ABB RAPID module: tester_right.mod

MODULE tester_right
LOCAL CONST string YuMi_App_Program_Version:="1.0.1"; !Do not edit or remove this line!
LOCAL VAR robtarget s35 := [[358.37,-68.33,133],[0.275214,0.0426853,0.863133,0.421233],[0,-2,-1,11],[-117.324,9E+09,9E+09,9E+09,9E+09,9E+09]];
LOCAL VAR robtarget s34 := [[537.58,-221.99,107.92],[0.0203865,-0.290011,-0.954645,-0.0642686],[0,-2,0,11],[-176.329,9E+09,9E+09,9E+09,9E+09,9E+09]];
LOCAL VAR robtarget s33 := [[467.55,-213.81,57.09],[0.496621,-0.80295,-0.0521253,-0.325456],[0,0,0,11],[165.649,9E+09,9E+09,9E+09,9E+09,9E+09]];
LOCAL VAR robtarget s32 := [[306.2,-52.91,16.67],[0.717218,-0.691447,0.0462227,-0.073234],[1,0,0,11],[153.702,9E+09,9E+09,9E+09,9E+09,9E+09]];
LOCAL VAR robtarget s31 := [[310.32,9.22,5.39],[0.716537,-0.693105,0.0533556,-0.0577434],[1,0,0,11],[153.592,9E+09,9E+09,9E+09,9E+09,9E+09]];
LOCAL VAR robtarget s30 := [[306.4,0.86,31.28],[0.734937,-0.673984,0.0222505,-0.0715334],[1,0,0,11],[152.628,9E+09,9E+09,9E+09,9E+09,9E+09]];
LOCAL VAR robtarget s29 := [[311.66,-63,44.82],[0.56004,-0.794065,-0.0460185,-0.231728],[0,0,0,11],[154.727,9E+09,9E+09,9E+09,9E+09,9E+09]];
LOCAL VAR robtarget s28 := [[299.07,-103.69,-6.2],[0.280816,-0.867914,-0.384884,-0.140468],[0,0,-1,11],[154.742,9E+09,9E+09,9E+09,9E+09,9E+09]];
LOCAL VAR robtarget s27 := [[352.75,-152.26,-47.58],[0.00513543,0.702291,0.711785,0.0111369],[1,0,-1,1010],[149.493,9E+09,9E+09,9E+09,9E+09,9E+09]];
LOCAL VAR robtarget s26 := [[345.22,-148.03,-90.26],[0.00526599,-0.716656,-0.697243,-0.0151133],[1,0,-1,1010],[153.525,9E+09,9E+09,9E+09,9E+09,9E+09]];
LOCAL VAR robtarget s25 := [[345.92,-149.32,-76.57],[0.0108524,-0.753223,-0.657389,-0.0194125],[1,0,-1,1010],[156.115,9E+09,9E+09,9E+09,9E+09,9E+09]];
LOCAL VAR robtarget s24 := [[357.66,-150.93,-35.49],[0.00970556,0.737723,0.663169,0.126002],[0,0,0,1010],[163.101,9E+09,9E+09,9E+09,9E+09,9E+09]];
LOCAL VAR robtarget s23 := [[388.73,-144.04,35.15],[0.0733127,-0.627707,-0.616071,-0.470176],[0,-1,0,11],[-163.98,9E+09,9E+09,9E+09,9E+09,9E+09]];
LOCAL VAR robtarget s22 := [[342.3,-148.5,49.05],[0.350551,-0.529329,-0.492073,-0.595641],[0,-1,0,11],[-159.838,9E+09,9E+09,9E+09,9E+09,9E+09]];
LOCAL VAR robtarget s21 := [[285.33,-50.36,-15.16],[0.467312,-0.523371,-0.473345,-0.532585],[0,-1,0,11],[-169.176,9E+09,9E+09,9E+09,9E+09,9E+09]];
LOCAL VAR robtarget s20 := [[284.5,11.38,-19.53],[0.493118,-0.506889,-0.461514,-0.535634],[1,-1,0,11],[-170.503,9E+09,9E+09,9E+09,9E+09,9E+09]];
LOCAL VAR robtarget s19 := [[284.5,11.39,-19.53],[0.49312,-0.506885,-0.461513,-0.535636],[1,-1,0,11],[-170.503,9E+09,9E+09,9E+09,9E+09,9E+09]];
LOCAL VAR robtarget s18 := [[283.93,11.08,-19.46],[0.493586,-0.506785,-0.461377,-0.535419],[1,-1,0,11],[-170.522,9E+09,9E+09,9E+09,9E+09,9E+09]];
LOCAL VAR robtarget s17 := [[283.93,11.07,-19.46],[0.493582,-0.506788,-0.461378,-0.535418],[1,-1,0,11],[-170.522,9E+09,9E+09,9E+09,9E+09,9E+09]];
LOCAL VAR robtarget s16 := [[283.93,11.07,-19.47],[0.493573,-0.5068,-0.461384,-0.53541],[1,-1,0,11],[-170.522,9E+09,9E+09,9E+09,9E+09,9E+09]];
LOCAL VAR robtarget s15 := [[282.43,12.65,-10.4],[0.493036,-0.507364,-0.460348,-0.536261],[1,-1,0,11],[-169.512,9E+09,9E+09,9E+09,9E+09,9E+09]];
LOCAL VAR robtarget s14 := [[285.29,11.12,13.96],[0.483333,-0.506561,-0.479515,-0.529009],[0,-1,0,11],[-167.842,9E+09,9E+09,9E+09,9E+09,9E+09]];
LOCAL VAR robtarget s13 := [[299.2,-72.45,52.01],[0.505778,-0.516645,-0.4521,-0.522371],[0,-1,0,11],[-163.463,9E+09,9E+09,9E+09,9E+09,9E+09]];
LOCAL VAR robtarget s12 := [[301.58,-60.87,67.73],[0.531821,-0.485612,-0.484682,-0.496418],[0,-1,0,11],[-162.383,9E+09,9E+09,9E+09,9E+09,9E+09]];
LOCAL VAR robtarget s11 := [[315.49,-68.53,58.63],[0.496532,-0.515442,-0.489328,-0.49833],[0,-1,0,11],[-161.717,9E+09,9E+09,9E+09,9E+09,9E+09]];
LOCAL VAR robtarget s10 := [[315.48,-68.53,58.63],[0.496531,-0.515444,-0.489327,-0.49833],[0,-1,0,11],[-161.717,9E+09,9E+09,9E+09,9E+09,9E+09]];
LOCAL VAR robtarget s9 := [[335.43,-129.87,89.3],[0.417557,-0.554213,-0.666307,-0.273002],[0,-1,0,11],[-161.728,9E+09,9E+09,9E+09,9E+09,9E+09]];
LOCAL VAR robtarget s8 := [[345.66,-189.94,55.79],[0.0163252,-0.262519,-0.955378,-0.134427],[0,-2,0,11],[-147.912,9E+09,9E+09,9E+09,9E+09,9E+09]];
LOCAL VAR robtarget s7 := [[253.69,-227.69,32.72],[0.0393185,-0.0503203,0.995728,-0.0666949],[0,-2,0,11],[-149.635,9E+09,9E+09,9E+09,9E+09,9E+09]];
LOCAL VAR robtarget s6 := [[285.53,-146.72,-90.22],[0.000644566,7.67705E-05,-0.999188,0.0402885],[0,-2,0,11],[-155.028,9E+09,9E+09,9E+09,9E+09,9E+09]];
LOCAL VAR robtarget s5 := [[285.55,-146.72,-90.22],[0.000628571,4.59053E-05,-0.999188,0.0402877],[0,-2,0,11],[-155.026,9E+09,9E+09,9E+09,9E+09,9E+09]];
LOCAL VAR robtarget s4 := [[285.56,-146.75,-90.22],[0.00061882,2.02596E-05,-0.999187,0.0403124],[0,-2,0,11],[-155.025,9E+09,9E+09,9E+09,9E+09,9E+09]];
LOCAL VAR robtarget s3 := [[283.94,-148.1,-80.96],[0.00559929,-0.00185021,0.999284,-0.0373822],[0,-2,0,11],[-154.675,9E+09,9E+09,9E+09,9E+09,9E+09]];
LOCAL VAR robtarget s2 := [[303.87,-127.03,37.37],[0.0164974,0.00923537,0.992408,0.12153],[0,-2,0,11],[-150.299,9E+09,9E+09,9E+09,9E+09,9E+09]];
LOCAL VAR robtarget s1 := [[358.37,-68.33,133],[0.275214,0.0426862,0.863132,0.421234],[0,-2,-1,11],[-117.324,9E+09,9E+09,9E+09,9E+09,9E+09]];
PROC main()
MoveSync s1;
OpenHand;
MoveSync s2;
MoveSync s3;
MoveSync s4;
MoveSync s5;
MoveSync s6;
CloseHand;
MoveSync s7;
MoveSync s8;
MoveSync s9;
MoveSync s10;
MoveSync s11;
MoveSync s12;
MoveSync s13;
MoveSync s14;
MoveSync s15;
MoveSync s16;
MoveSync s17;
MoveSync s18;
MoveSync s19;
MoveSync s20;
OpenHand;
MoveSync s21;
MoveSync s22;
MoveSync s23;
MoveSync s24;
MoveSync s25;
MoveSync s26;
CloseHand;
MoveSync s27;
MoveSync s28;
MoveSync s29;
MoveSync s30;
MoveSync s31;
OpenHand;
MoveSync s32;
MoveSync s33;
MoveSync s34;
MoveSync s35;
ENDPROC
ENDMODULE
